(* PLC project Generated.project, CODESYS CODESYS V3.5 SP19 Patch 1 *)
(* stored: creationDateTime 2026-11-18T02:47:08.643597, modificationDateTime 2026-11-18T02:47:08.643597 *)

(* ======================================================================= ⚙️ ST_fbMachineHomingCycle_Cfg — Réglages de FB_CycleMachineHoming ─────────────────────────────────────────────────────────────────────── 🎯 Rôle : Réglages géométriques du référencement machine (cible haute M2/benne + écarts benne) + temporisations de garde du GRAFCET de homing (montée, homing axes). 🔒 Ownership : produit par PRG_02_Acquisition depuis _WinchM2CfgPersist (cible haute) et _BucketCfgPersist (écarts, GVL_PERSISTENT). Initialized : drapeau de restauration boot (pont persistant). 📄 Doc métier : DOC/AF/AF_Partie-09_Fonction_Encoder_v2.4.md (F09.08) ======================================================================= *)
TYPE ST_fbMachineHomingCycle_Cfg : STRUCT
  CfgTopHomingTarget_M : REAL;  (* Position capteur haut M2/benne (m) — cible finale HX4 M2 (+ OffsetCloseM) *)
  CfgTopHomingTargetM1_M : REAL := 8.5;  (* Position capteur haut M1 (m) — cible finale HX4 M1 (defaut 8.5 m) *)
  CfgOffsetOpen_M : REAL;  (* Ecart géométrique benne ouverte (m) *)
  CfgOffsetClose_M : REAL;  (* Ecart géométrique benne fermée (m) *)
  CfgTimeoutClimb : TIME := TIME#300s0ms;  (* Garde de montee : budget d'une MONTER CONTINUE (un temporisateur remet son temps ecoule a zero des que la commande retombe : une pause operateur ou un arret d'urgence ne consomme donc rien). Derivation : course maximale de cable = CfgTopSensorPos_M - CfgCableLimitDescent_M (8,5 m - (-50 m) = 58,5 m) ; borne haute de vitesse du palier 1 = 0,4 m/s (GVL_PERSISTENT._WinchSpeedConfig.SpeedBandMaxMps[1], valeur de banc A MESURER sur site) => 58,5 / 0,4 = 146,3 s ; marge x2 = 292,5 s ; valeur retenue 300 s (arrondie au-dessus). A revoir si la course ou la vitesse du palier 1 changent (gate G511). Garde de montee au capteur haut (0 = pas de garde) *)
  CfgEntryHoldTime : TIME := TIME#5s0ms;  (* Duree maintien BP joystick au neutre en HX0 (MAINT_N1) *)
  CfgBucketPrepareTimeout : TIME := TIME#20s0ms;  (* Duree max commande continue M2 en HX1 (coupe -> neutre) *)
  CfgSlackReliefMaxTime : TIME := TIME#2s0ms;  (* Duree max descente detente cable par geste en HX2 *)
  CfgTopClearanceTime : TIME := TIME#4s0ms;  (* Duree descente accumulee apres relachement TOP en HX3 *)
  CfgTimeoutHomeAxes : TIME := TIME#60s0ms;  (* Garde globale prise de reference (HX4) *)
  Initialized : BOOL := FALSE;  (* Drapeau de restauration config au boot (pont persistant) *)
END_STRUCT;
END_TYPE
